{attribute addProperty BoxType "EL6201-0000-0017"}
{attribute addProperty Id "Slave_13A_DI0BIT10.12597Slave_13A_DI1BIT10.12598Slave_13A_DI2BIT10.12599Slave_13A_DI3BIT10.125100Slave_13B_DI0BIT10.125101Slave_13B_DI1BIT10.125102Slave_13B_DI2BIT10.125103Slave_13B_DI3BIT10.125104"}
{attribute addProperty CRC "1542086936"}
{attribute addProperty SizeInBites "8"}
{attribute addProperty SizeInBytes "1"}
TYPE Slave_13_Inputs_5BEA6118 :
STRUCT
	{attribute addProperty Name "Slave_13A_DI0"}
	Slave_13A_DI0 : BIT;
	{attribute addProperty Name "Slave_13A_DI1"}
	Slave_13A_DI1 : BIT;
	{attribute addProperty Name "Slave_13A_DI2"}
	Slave_13A_DI2 : BIT;
	{attribute addProperty Name "Slave_13A_DI3"}
	Slave_13A_DI3 : BIT;
	{attribute addProperty Name "Slave_13B_DI0"}
	Slave_13B_DI0 : BIT;
	{attribute addProperty Name "Slave_13B_DI1"}
	Slave_13B_DI1 : BIT;
	{attribute addProperty Name "Slave_13B_DI2"}
	Slave_13B_DI2 : BIT;
	{attribute addProperty Name "Slave_13B_DI3"}
	Slave_13B_DI3 : BIT;
END_STRUCT
END_TYPE

(* stored: Version 1.2.0.0, ProductVersion 3.1.4024.9
   DUT Slave_13_Inputs_5BEA6118: Id {16e9f8ad-1dc9-4d23-a020-13b35436a0f0} *)
